Fanuc KAREL source: GET_POS_REG.kl

PROGRAM T
%NOLOCKGROUP
VAR
 v0 : INTEGER
 v1 : INTEGER
 v2 : INTEGER
 res : XYZWPREXT
BEGIN
 res = GET_POS_REG(v0, v1, v2)
END T
